(* PLC project Tc2_Utilities.F_SplitBIC Demo, tc3-libraries-kb TwinCAT 3.1 *)
(* stored: creationDateTime 2026-05-10T19:00:00, modificationDateTime 2026-05-10T19:00:00 *)

PROGRAM P_Demo_F_SplitBIC
  VAR
    rResult : ST_SplittedBIC;  (* F_SplitBIC 返回值 *)
    bRun : BOOL;  (* 触发一次调用 *)
    sBIC : STRING := '1P193995SBTN0002agdw1KEL7411 Q1 2P112104020018';  (* 测试用本地变量 *)
  END_VAR

            // ============================================================
// Tc2_Utilities.F_SplitBIC 演示程序（FUNCTION）
// ============================================================
// 验证步骤：
//   1. 引用 Tc2_Utilities
//   2. 编译 + 登录
//   3. 强制 bRun := TRUE 一个周期
//   4. 在线监视 rResult / 各 demo 变量
// ============================================================

IF bRun THEN
    rResult := F_SplitBIC(sBIC);
    bRun := FALSE;
END_IF;

          
END_PROGRAM
